Staubli VAL3: util.dtx

num nTest
public bool bDebug
public mdesc mNomSpeed = {blend=off}
